// TwinCAT 3 PLC project PLC_NoveltyDetection
// ProgramVersion: 3.1.4024.0
// libraries:
//   Tc2_Standard, * (Beckhoff Automation GmbH)
//   Tc2_System, * (Beckhoff Automation GmbH)
//   Tc3_Module, * (Beckhoff Automation GmbH)
//   Tc3_Vision, * (Beckhoff Automation GmbH)
// project tree:
//   DUTs/ E_NoveltyDetectorType.TcDUT, ST_NoveltyDetectorParams.TcDUT
//   / PlcTask.TcTTO
//   POUs/ FB_TrainingDataHandler.TcPOU, F_ExtractFeatures.TcPOU, MAIN.TcPOU
// real-time tasks:
//   TASK PlcTask: cycle T#10ms, priority 20, ADS port 350
//   TASK VnTask ImgAcq (TrainingImages): cycle T#10ms, priority 5, ADS port 351
//   TASK VnTask ImgAcq (TestImages): cycle T#10ms, priority 6, ADS port 352

CONFIGURATION PLC_NoveltyDetection
    RESOURCE PLC ON TwinCAT3
        TASK PlcTask(INTERVAL := T#10ms, PRIORITY := 20);
        PROGRAM MAIN WITH PlcTask : MAIN;
    END_RESOURCE
END_CONFIGURATION

// ---- DUTs/E_NoveltyDetectorType.TcDUT
{attribute 'qualified_only'}
{attribute 'strict'}
TYPE E_NoveltyDetectorType :
(
	KMPP := 0,
	KNN,
	LBG,
	NBC,
	STA,
	SVM
);
END_TYPE

// ---- DUTs/ST_NoveltyDetectorParams.TcDUT
TYPE ST_NoveltyDetectorParams :
STRUCT
	nKmppK					:	UDINT 				:=	2;
	bKmppDoublePrecision	:	BOOL 				:=	FALSE;		// optional Exp parameter
	nKmppMaxIterations		:	UDINT				:=	10;			// optional Exp parameter
	fKmppEpsilon			:	LREAL				:=	0.001;		// optional Exp parameter
	nKnnK					:	UDINT 				:=	1;
	nLbgMaxClusters			:	UDINT				:=	5;
	fLbgMaxClusterRadius	:	LREAL				:=	1.0;
	bLbgSingleSplitSteps	:	BOOL				:=	TRUE;
	bLbgDoublePrecision		:	BOOL				:=	FALSE;		// optional Exp parameter
	nLbgMaxIterations		:	UDINT				:=	10;			// optional Exp parameter
	fLbgEpsilon				:	LREAL				:=	0.001;		// optional Exp parameter
	fStaRho	                :	LREAL				:=	0.73;
	nStaNu	                :	UDINT				:=	5;			// optional Exp parameter
	bStaDoublePrecision		:	BOOL				:=	TRUE;		// optional Exp parameter
	fStaBetaSbm				:	LREAL				:=	0.0;		// optional Exp parameter
	nStaPhi					:	UDINT				:=	1;			// optional Exp parameter
	nStaTau					:	UDINT				:=	100;		// optional Exp parameter	
	fSvmNu					:	LREAL				:=	0.4;		// 0.4 Apple or 0.5 Banane
	eSvmKernelType			:	ETcVnSvmKernelType	:=	ETcVnSvmKernelType.TCVN_SKT_RBF;
	fSvmGamma				:	LREAL				:=	0.000001;
	fSvmCoef0				:	LREAL				:=	0;
	fSvmDegree				:	LREAL				:=	0;
	nSvmMaxIterations		:	UDINT				:=	100000;		// optional Exp parameter
	fSvmEpsilon				:	LREAL				:=	0.0001;		// optional Exp parameter
END_STRUCT
END_TYPE

// ---- POUs/MAIN.TcPOU
PROGRAM MAIN
VAR
	eNoveltyDetectorType: 	E_NoveltyDetectorType;		// Novelty detector type
	stParams			:	ST_NoveltyDetectorParams;	// Novelty detector parameters
	bResetModel			:	BOOL;						// Reset model to start a new training with a changed model or parameters
	bResetTrainingData	:	BOOL;						// Reset the trained features to get new ones and train model
	eTrainedModelType	: 	E_NoveltyDetectorType;
	
	hrTrain				:	HRESULT;
	hrTest				:	HRESULT;
	
	ipImageTest			:	ITcVnImage;
	ipImageResDisp		:	ITcVnDisplayableImage;
	
	eCameraState		:	ETcVnCameraState;	
	fbCameraTest		:	FB_VN_SimpleCameraControl;
	
	fbTrainingDataHandler:	FB_TrainingDataHandler;
	
	ipNoveltyDetectorModel:	ITcVnMlModel;
	ipSamplesTraining	:	ITcVnContainer;
	ipFeatureScaling	:	ITcVnContainer;
	ipSampleTest		:	ITcVnContainer;
	fNovelty			:	REAL;
	
	// Result
	fNoveltyThreshold	:	REAL;
	sLabel				:	STRING(255);
	aGreen				:	TcVnVector4_LREAL := [0, 255, 0];
END_VAR

// Disclaimer

// This publication contains statements about the suitability of our products for certain
// areas of application. These statements are based on typical features of our products.
// The examples shown in this publication are for demonstration purposes only.
// The information provided herein should not be regarded as specific operation characteristics.
// It is incumbent on the customer to check and decide whether a product is suitable for use
// in a particular application. We do not give any warranty that the source code which is
// made available with this publication is complete or accurate.

// THE SAMPLE CODE CONTAINED IN THIS PUBLICATION IS PROVIDED “AS IS” WITHOUT WARRANTY OF ANY KIND,
// EITHER EXPRESSED, IMPLIED OR STATUTORY, INCLUDING WITHOUT LIMITATION, ANY WARRANTY WITH RESPECT TO NON-INFRINGEMENT,
// FREEDOM FROM PROPRIETARY RIGHTS OF THIRD PARTIES OR FITNESS FOR ANY PARTICULAR PURPOSE.

// This publication may be changed from time to time without prior notice.
// No liability is assumed for errors and/or omissions.
// Our products are described in detail in our data sheets and documentations.
// Product-specific warnings and cautions must be observed.
// For the latest version of our data sheets and documentations visit our website (www.beckhoff.de).

// © Beckhoff Automation GmbH & Co. KG, December 2023

// The reproduction, distribution and utilization of this document as well as the communication
// of its contents to others without express authorization is prohibited. 
// Offenders will be held liable for the payment of damages.
// All rights reserved in the event of the grant of a patent, utility model or design.

//	==========================================================================================

// SAMPLE - Machine Learning Novelty (Anomaly) Detection
//	-------------------------------------------------------

// Steps To Do:
// ------------
// 1. Add the training images to the TrainingImages control, only the images of one object class can be selected
// 2. Add the test images to the TestingImages control
// 3. Activate the configuration -> Start TwinCAT system and PLC to run -> watch the results in the ADS Image Watch
// 4. Change eNoveltyDetectorType and stParams to change the model or settings
// 5. Set bResetModel to start create a new model and start training
//    Note: If you change to eClassifierType = STA or from this type to another, a bResetTrainingData is automatically performed due to the different scaling of the training data.
// 6. Set bResetTrainingData to get new training data if images or feature extraction changed

// Reset the trained features to get new ones and train model
IF bResetTrainingData
	OR (eTrainedModelType <> E_NoveltyDetectorType.STA AND eNoveltyDetectorType = E_NoveltyDetectorType.STA)
	OR (eTrainedModelType = E_NoveltyDetectorType.STA AND eNoveltyDetectorType <> E_NoveltyDetectorType.STA) THEN
	
	bResetTrainingData := FALSE;
	fbTrainingDataHandler.Reset();
	FW_SafeRelease(ADR(ipSamplesTraining));
	FW_SafeRelease(ADR(ipFeatureScaling));
	FW_SafeRelease(ADR(ipNoveltyDetectorModel));
	eTrainedModelType := eNoveltyDetectorType;
	// Reset return value
	hrTrain := S_OK;
END_IF

// Get sample data for training
fbTrainingDataHandler(eNoveltyDetectorType := eNoveltyDetectorType);
IF ipSamplesTraining = 0 AND ipFeatureScaling = 0 THEN
	hrTrain := fbTrainingDataHandler.GetTrainingData(ipSamplesTraining, ipFeatureScaling);
END_IF

// Retrain with changed model or parameters
IF bResetModel THEN
	bResetModel := FALSE;
	FW_SafeRelease(ADR(ipNoveltyDetectorModel));
	eTrainedModelType := eNoveltyDetectorType;
	// Reset return value
	hrTrain := S_OK;
END_IF

IF SUCCEEDED(hrTrain) AND ipSamplesTraining <> 0 AND ipNoveltyDetectorModel = 0 THEN

// Set novelty threshold according to model results 
fNoveltyThreshold := 1.0;
			
	// Create the model
	CASE eNoveltyDetectorType OF
		
		E_NoveltyDetectorType.KMPP:
			hrTrain := F_VN_CreateKmppModelExp(
							ipMlModel			:=	ipNoveltyDetectorModel,
							eKmppType			:=	TCVN_PC_NOVELTY_DETECTOR,
							nK					:=	stParams.nKmppK,
							bDoublePrecision	:=	stParams.bKmppDoublePrecision,
							nMaxIterations		:=	stParams.nKmppMaxiterations,
							fEpsilon			:=	stParams.fKmppEpsilon,
							hrPrev				:=	hrTrain);
		
		E_NoveltyDetectorType.KNN:
			hrTrain := F_VN_CreateKnnModel(
							ipMlModel			:=	ipNoveltyDetectorModel,
							eKnnType			:=	TCVN_KNN_NOVELTY_DETECTOR,
							nK					:=	stParams.nKnnK,
							hrPrev				:=	hrTrain);
			
		E_NoveltyDetectorType.LBG:
			hrTrain := F_VN_CreateLbgModelExp(
							ipMlModel			:=	ipNoveltyDetectorModel,
							eLbgType			:=	TCVN_PC_NOVELTY_DETECTOR,
							nMaxClusters		:=	stParams.nLbgMaxClusters,
							fMaxClusterRadius	:=	stParams.fLbgMaxClusterRadius,
							bSingleSplitSteps	:=	stParams.bLbgSingleSplitSteps,
							bDoublePrecision	:=	stParams.bLbgDoublePrecision,
							nMaxiterations		:=	stParams.nLbgMaxIterations,
							fEpsilon			:=	stParams.fLbgEpsilon,
							hrPrev				:=	hrTrain);
			
		E_NoveltyDetectorType.NBC:
			hrTrain := F_VN_CreateNbcModel(
							ipMlModel			:=	ipNoveltyDetectorModel,
							eNbcType			:=	TCVN_NBC_NOVELTY_DETECTOR,
							hrPrev				:=	hrTrain);
							
			// Set novelty threshold according to model results 
			fNoveltyThreshold := 4.0;							

		E_NoveltyDetectorType.STA:
			hrTrain := F_VN_CreateStaModelExp2(
							ipMlModel           :=	ipNoveltyDetectorModel,
							eStaType            :=	TCVN_STA_NOVELTY_DETECTOR,
							fRho                :=	stParams.fStaRho,
							nNu                 :=	stParams.nStaNu,
							bDoublePrecision    :=	stParams.bStaDoublePrecision,
							fBetaSbm			:=	stParams.fStaBetaSbm,
							nPhi				:=	stParams.nStaPhi,
							nTau				:=	stParams.nStaTau,
							hrPrev				:=	hrTrain);
								
			// Set novelty threshold according to model results 
			fNoveltyThreshold := 0.3;
		
		E_NoveltyDetectorType.SVM:
			hrTrain := F_VN_CreateSvmModelExp(
							ipMlModel			:=	ipNoveltyDetectorModel,
							eSvmType			:=	TCVN_SVM_NOVELTY_DETECTOR,
							fC					:=	0,
							fNu					:=	stParams.fSvmNu,
							fP					:=	0,
							eKernelType			:=	stParams.eSvmKernelType,
							fGamma				:=	stParams.fSvmGamma,
							fCoef0				:=	stParams.fSvmCoef0,
							fDegree				:=	stParams.fSvmDegree,
							nMaxIterations		:=	stParams.nSvmMaxIterations,
							fEpsilon			:=	stParams.fSvmEpsilon,
							hrPrev				:=	hrTrain);
	
	END_CASE
	
	// Train model
	hrTrain := F_VN_TrainBatch(
					ipMlModel   :=  ipNoveltyDetectorModel,
					ipSamples   :=  ipSamplesTraining,
					ipOutputs   :=  0,
					hrPrev      :=  hrTrain);

END_IF

// Get test images
eCameraState := fbCameraTest.GetState();

IF eCameraState = TCVN_CS_ERROR THEN
	hrTest := fbCameraTest.Reset();

ELSIF eCameraState < TCVN_CS_ACQUIRING THEN
	hrTest := fbCameraTest.StartAcquisition();

// Camera streaming
ELSIF eCameraState = TCVN_CS_ACQUIRING THEN
	hrTest := fbCameraTest.GetCurrentImage(ipImageTest);

	// Check if new image was received
	IF SUCCEEDED(hrTest) AND ipImageTest <> 0 THEN

        IF ipNoveltyDetectorModel <> 0 AND ipFeatureScaling <> 0 THEN
			// Get features from sample image and scale 
			hrTest := F_ExtractFeatures(ipImageTest, ipSampleTest, hrTest);
			IF  eNoveltyDetectorType = E_NoveltyDetectorType.STA THEN
				hrTest := F_VN_FeatureScalingExp(ipSampleTest, ipFeatureScaling, ipSampleTest, 0.2, 0.8, hrTest);
			ELSE
				hrTest := F_VN_FeatureScaling(ipSampleTest, ipFeatureScaling, ipSampleTest, hrTest);
			END_IF
			
			// Get novelty result
			hrTest := F_VN_GetSampleNovelty(ipNoveltyDetectorModel, ipSampleTest, fNovelty, hrTest);
			
			// Check the degree of novelty and write result
			IF fNovelty <= fNoveltyThreshold THEN
				sLabel := CONCAT('Known: ',REAL_TO_STRING(fNovelty));
			ELSE
				sLabel := CONCAT('Unknown: ',REAL_TO_STRING(fNovelty));
			END_IF
			hrTest := F_VN_PutTextExp(sLabel, ipImageTest, 30, 60, TCVN_FT_HERSHEY_PLAIN, 4, aGreen, 2, TCVN_LT_ANTIALIASED, FALSE, hrTest);
		END_IF
		
		// Display image
		hrTest := F_VN_TransformIntoDisplayableImage(ipImageTest, ipImageResDisp, S_OK);
	END_IF
END_IF

END_PROGRAM

// ---- POUs/FB_TrainingDataHandler.TcPOU
FUNCTION_BLOCK PUBLIC FB_TrainingDataHandler
VAR_INPUT
	 eNoveltyDetectorType : E_NoveltyDetectorType;
END_VAR
VAR_OUTPUT
END_VAR
VAR
	hr					: HRESULT;
	eCameraState		: ETcVnCameraState;
	fbCameraTraining	: FB_VN_SimpleCameraControl;	
	ipImageTraining		: ITcVnImage;
	ipImageTrainingDisp	: ITcVnDisplayableImage;
	bTrigger			: BOOL := TRUE;
	sLabel				: STRING(255);
	aGreen				: TcVnVector4_LREAL := [0, 255, 0];
	
	// Image Info
	nImagesTotal		: UDINT := 6;
	nImagesLoaded		: UDINT := 0;
	
	ipFeatures			: ITcVnContainer;
	ipImageFeatures		: ITcVnContainer;
	ipScales			: ITcVnContainer;
	ipScaledFeatures	: ITcVnContainer;
END_VAR

// Initialize container
IF ipImageFeatures = 0 THEN
	hr := F_VN_CreateContainer(ipImageFeatures, ContainerType_Vector_Vector_LREAL, nImagesTotal, hr);
END_IF

// Get training images
eCameraState := fbCameraTraining.GetState();

IF eCameraState = TCVN_CS_ERROR THEN
	hr := fbCameraTraining.Reset();
	
// Camera trigger image
ELSIF eCameraState = TCVN_CS_TRIGGERING THEN
	hr := fbCameraTraining.TriggerImage();
	
ELSIF eCameraState < TCVN_CS_ACQUIRING THEN
	hr := fbCameraTraining.StartAcquisition();

// Camera streaming
ELSIF eCameraState = TCVN_CS_ACQUIRING THEN

	IF bTrigger THEN
		hr := fbCameraTraining.TriggerImage();
		IF SUCCEEDED(hr) THEN
			bTrigger := FALSE;
		END_IF
	ELSE
		hr := fbCameraTraining.GetCurrentImage(ipImageTraining);

		// Check if new image was received
		IF SUCCEEDED(hr) AND ipImageTraining <> 0 THEN
			
			// Get features from training image 
			hr := F_ExtractFeatures(ipImageTraining, ipFeatures, hr);
		
			// Add features to the container
			hr := F_VN_SetAt_ITcVnContainer(ipFeatures, ipImageFeatures, nImagesLoaded, hr);
			FW_SafeRelease(ADR(ipFeatures));
			
			// Display image
			sLabel := CONCAT('Image Number: ', UDINT_TO_STRING(nImagesLoaded + 1));
			hr := F_VN_PutTextExp(sLabel, ipImageTraining, 30, 60, TCVN_FT_HERSHEY_PLAIN, 4, aGreen, 2, TCVN_LT_ANTIALIASED, FALSE, hr);
			hr := F_VN_TransformIntoDisplayableImage(ipImageTraining, ipImageTrainingDisp, hr);
			
			nImagesLoaded := nImagesLoaded + 1;
			IF nImagesLoaded < nImagesTotal THEN
				// Trigger next image
				bTrigger := TRUE;
			ELSE
				// After collecting all training data, normalize the feature values
				hr := F_VN_GetFeatureScales(ipImageFeatures, ipScales, TCVN_FST1_MINMAX, hr);
				IF  eNoveltyDetectorType = E_NoveltyDetectorType.STA THEN
					hr := F_VN_FeatureScalingExp(ipImageFeatures, ipScales, ipScaledFeatures, 0.2, 0.8, hr);
				ELSE
					hr := F_VN_FeatureScaling(ipImageFeatures, ipScales, ipScaledFeatures, hr);
				END_IF
				FW_SafeRelease(ADR(ipImageFeatures));
			END_IF
		END_IF
	END_IF
END_IF

METHOD PUBLIC GetTrainingData : HRESULT
VAR_INPUT
	ipTrainingSamples	: REFERENCE TO ITcVnContainer;
	ipFeatureScaling	: REFERENCE TO ITcVnContainer;
END_VAR
VAR
	hr					: HRESULT;
END_VAR
IF nImagesLoaded = nImagesTotal THEN
	hr := F_VN_CopyContainer(ipScaledFeatures, ipTrainingSamples, hr);
	GetTrainingData := F_VN_CopyContainer(ipScales, ipFeatureScaling, hr);
ELSE
	GetTrainingData := S_PENDING;
END_IF
END_METHOD

METHOD PUBLIC Reset : HRESULT
VAR_INPUT
END_VAR
nImagesLoaded := 0;
FW_SafeRelease(ADR(ipFeatures));
FW_SafeRelease(ADR(ipImageFeatures));
FW_SafeRelease(ADR(ipScales));
FW_SafeRelease(ADR(ipScaledFeatures));
bTrigger := TRUE;
END_METHOD

END_FUNCTION_BLOCK

// ---- POUs/F_ExtractFeatures.TcPOU
FUNCTION F_ExtractFeatures : HRESULT
VAR_INPUT
	ipImage		:	ITcVnImage;
	ipFeatures	:	REFERENCE TO ITcVnContainer;
	hrPrev		:	HRESULT;
END_VAR
VAR
	hr			:	HRESULT;
	aAverage	:	TcVnVector4_LREAL;
	aFeatures	:	ARRAY [0..2] OF LREAL;
END_VAR

IF FAILED(hrPrev) THEN
	F_ExtractFeatures := hrPrev;
	RETURN;
END_IF

IF ipImage = 0 THEN
	F_ExtractFeatures := Tc2_System.E_HRESULTAdsErr.INVALIDPARM;
	RETURN;
END_IF

// Simple feature extraction example 
hr := F_VN_ImageAverage(ipImage, aAverage, hr);

aFeatures[0] := aAverage[0];
aFeatures[1] := aAverage[1];
aFeatures[2] := aAverage[2];

// Create a container with all features as a vector
hr := F_VN_CreateContainerFromArray(ADR(aFeatures), ipFeatures, ContainerType_Vector_LREAL, 3, hr);

F_ExtractFeatures := hr;

END_FUNCTION
